// TwinCAT 3 PLC project MAS418_PLC2
// ProgramVersion: 3.1.4023.0
// libraries:
//   Tc2_Standard, * (Beckhoff Automation GmbH)
//   Tc2_System, * (Beckhoff Automation GmbH)
//   Tc3_Module, * (Beckhoff Automation GmbH)
// project tree:
//   Task1/ G_task1.TcGVL, P_task1.TcPOU, Sensors.TcDUT
//   / PlcTask.TcTTO
//   POUs/ MAIN.TcPOU
//   Task2/ fDeg2Rad.TcPOU, ST_Timer.TcDUT, g_task2.TcGVL, p_task2.TcPOU
//   Task3/ E_StateMachine.TcDUT, F_UpdatePara2.TcPOU, g_task3.TcGVL, F_UpdatePara.TcPOU, p_task3.TcPOU, ST_MotorPara.TcDUT
// real-time tasks:
//   TASK PlcTask: cycle T#10ms, priority 20, ADS port 350

CONFIGURATION MAS418_PLC2
    RESOURCE PLC ON TwinCAT3
        TASK PlcTask(INTERVAL := T#10ms, PRIORITY := 20);
        PROGRAM MAIN WITH PlcTask : MAIN;
    END_RESOURCE
END_CONFIGURATION

// ---- Task1/Sensors.TcDUT
{attribute 'qualified_only'}
{attribute 'strict'}
TYPE Sensors :
(
	Sick,
	Pilz,
	Parker,
	Bosch
);
END_TYPE

// ---- Task2/ST_Timer.TcDUT
TYPE ST_Timer :
STRUCT
	bTimerStart : BOOL; 
	tTimer : TIME; 
	bTimerOn : BOOL;
	tElapsedTime : TIME; 
END_STRUCT
END_TYPE

// ---- Task3/E_StateMachine.TcDUT
{attribute 'qualified_only'}
{attribute 'strict'}
TYPE E_StateMachine :
(
	State1,
	State2,
	State3

);
END_TYPE

// ---- Task3/ST_MotorPara.TcDUT
TYPE ST_MotorPara :
STRUCT
	fMax : REAL;
	fMin : REAL;
END_STRUCT
END_TYPE

// ---- Task1/G_task1.TcGVL
{attribute 'qualified_only'}
VAR_GLOBAL
	dtCurrentDt : DATE_AND_TIME := DT#2023-02-07-14:00:00;
	tTime : TIME := T#5S;
	aArray : ARRAY[1..4] OF DATE := [D#2023-02-07, D#2023-02-08, D#2023-02-09, D#2023-02-10];
	eSensor1 : Sensors;
	
    bTimerStart : BOOL; 
	tTimer : TIME := T#10S; 
	bTimerOn : BOOL;
	tElapsedTime : TIME; 
END_VAR

// ---- Task2/g_task2.TcGVL
{attribute 'qualified_only'}
VAR_GLOBAL
	stTimer2 : ST_Timer := (tTimer := T#5S);
	fAngPosM1deg : REAL;
	fAngPosM1rad : REAL;
END_VAR

// ---- Task3/g_task3.TcGVL
{attribute 'qualified_only'}
VAR_GLOBAL
	fNewParameter : REAL;
	stMotorPara : ST_MotorPara;
	stMotorPara2 : ST_MotorPara;
END_VAR

// ---- POUs/MAIN.TcPOU
PROGRAM MAIN
VAR
	bEnable : BOOL;
	bStart : BOOL;
END_VAR

bEnable:=bStart;
P_task1();
p_task2();
p_task3();

END_PROGRAM

// ---- Task1/P_task1.TcPOU
PROGRAM P_task1
VAR
	pPointer : POINTER TO DATE_AND_TIME := ADR(G_task1.dtCurrentDt);
	tReference : REFERENCE TO TIME REF=G_task1.tTime; 
	fbTon : TON;
END_VAR

pPointer^ := DT#2023-02-08-15:31:19;
tReference := T#20S;
G_task1.aArray[3] := D#2023-02-28;
G_task1.eSensor1 := Sensors.Bosch;

fbTon(
	IN := G_task1.bTimerStart, 
	PT := G_task1.tTimer,
	ET => G_task1.tElapsedTime,
	Q => G_task1.bTimerOn
);

END_PROGRAM

// ---- Task2/p_task2.TcPOU
PROGRAM p_task2
VAR
	fbTOF : TOF;
	
END_VAR

fbTOF(
	IN := g_task2.stTimer2.bTimerStart,
	PT := g_task2.stTimer2.tTimer,
	ET => g_task2.stTimer2.tElapsedTime,
	Q => g_task2.stTimer2.bTimerOn
);

g_task2.fAngPosM1rad := fDeg2Rad(g_task2.fAngPosM1deg);

END_PROGRAM

// ---- Task2/fDeg2Rad.TcPOU
FUNCTION fDeg2Rad : REAL
VAR_INPUT
	fDeg : LREAL;
END_VAR
VAR
	
END_VAR

fDeg2Rad := fDeg * (3.14/180);

END_FUNCTION

// ---- Task3/p_task3.TcPOU
PROGRAM p_task3
VAR
	fbRTrig : R_TRIG;
	bUpdateSpeed : BOOL;
	fNewValue : REAL;
	
	eStateMachine 	: E_StateMachine; 
	bEnable 		: BOOL;
	bStart 			: BOOL;
	bStop 			: BOOL;
END_VAR

fbRTrig(CLK := bUpdateSpeed);


F_UpdatePara(bUpdateValue := fbRTrig.Q, fNewValue :=  fNewValue, stMotorPara := g_task3.stMotorPara);

F_UpdatePara2(bUpdateValue := fbRTrig.Q, fNewValue :=  fNewValue, stMotorPara := g_task3.stMotorPara2);


CASE eStateMachine OF
	E_StateMachine.State1: 
		IF bEnable THEN
			eStateMachine := E_StateMachine.State2;
		END_IF
		
	E_StateMachine.State2: 
		IF NOT(bEnable) OR bStop THEN
			eStateMachine := E_StateMachine.State1;
		ELSIF bStart THEN
			eStateMachine := E_StateMachine.State3;
		END_IF
		
	E_StateMachine.State3: 
		IF NOT(bEnable) OR bStop THEN
			eStateMachine := E_StateMachine.State1;
		END_IF
ELSE 
	eStateMachine := E_StateMachine.State1;
END_CASE

END_PROGRAM

// ---- Task3/F_UpdatePara.TcPOU
FUNCTION F_UpdatePara : REAL
VAR_INPUT
	bUpdateValue : BOOL;
	fNewValue : REAL;
	stMotorPara : ST_MotorPara;
	
END_VAR
VAR
END_VAR

IF bUpdateValue THEN
	stMotorPara.fMax := fNewValue;
ELSE 
	stMotorPara.fMax := stMotorPara.fMax;	
END_IF

END_FUNCTION

// ---- Task3/F_UpdatePara2.TcPOU
FUNCTION F_UpdatePara2 : REAL
VAR_INPUT
	bUpdateValue : BOOL;
	fNewValue : REAL;
	stMotorPara : REFERENCE TO ST_MotorPara;
	
END_VAR
VAR
END_VAR

IF bUpdateValue THEN
	stMotorPara.fMax := fNewValue;
ELSE 
	stMotorPara.fMax := stMotorPara.fMax;	
END_IF

END_FUNCTION
